{attribute 'no_explicit_call' := 'do not call this FB directly'}{attribute 'enable_dynamic_creation'}
FUNCTION_BLOCK OutputPort_ANY EXTENDS Disposable IMPLEMENTS I_OutputPort
VAR
	_name : T_MAXSTRING;
	_dataType : T_MAXSTRING;
	internalBuffer : POINTER TO BYTE;
	internalBufferSize : UDINT;
	eventEmitter : EventEmitter;
END_VAR

METHOD PUBLIC Accept
VAR_INPUT
	Visitor : I_OutputPortVisitor;
END_VAR
Visitor.VisitOutputPort(this^);
END_METHOD

METHOD PRIVATE CopyInternalBufferToDestination
VAR_INPUT
	DestinationAddress : PVOID;
END_VAR
memcpy(DestinationAddress,internalBuffer,internalBufferSize);
END_METHOD

METHOD PRIVATE CopySourceToInternalBuffer
VAR_INPUT
	SourceAddress : PVOID;
END_VAR
memcpy(internalBuffer,SourceAddress,internalBufferSize);
END_METHOD

PROPERTY PUBLIC DataSize : UDINT
GET
IF internalBuffer = 0 THEN
	RETURN;
END_IF

DataSize := internalBufferSize;
END_GET
END_PROPERTY

PROPERTY PUBLIC DataType : T_MAXSTRING
GET
DataType := _dataType;
END_GET
END_PROPERTY

METHOD PRIVATE DeleteInternalBuffer
IF internalBuffer <> 0 THEN
	__DELETE(internalBuffer);
END_IF
END_METHOD

METHOD PRIVATE EmitOnOutputPortChangeEvent
VAR_INPUT
	PortChanged : I_OutputPort;
END_VAR
VAR
	pOutputPortChangeEvent : POINTER TO OutputPortChangedEvent;
END_VAR
pOutputPortChangeEvent := __NEW(OutputPortChangedEvent(TargetOutputPort := PortChanged));
eventEmitter.Emit('OnOutputPortChanged',pOutputPortChangeEvent^);
pOutputPortChangeEvent^.Dispose();
END_METHOD

METHOD FB_exit : BOOL
VAR_INPUT
	bInCopyCode : BOOL; // if TRUE, the exit method is called for exiting an instance that is copied afterwards (online change).
END_VAR
IF bInCopyCode THEN
	RETURN;
END_IF

DeleteInternalBuffer();
END_METHOD

METHOD FB_init : BOOL
VAR_INPUT
	bInitRetains : BOOL; // if TRUE, the retain variables are initialized (warm start / cold start)
	bInCopyCode : BOOL;  // if TRUE, the instance afterwards gets moved into the copy code (online change)
	Name : T_MAXSTRING;
	DataType : T_MAXSTRING;
	Parent : I_HaveOutputPorts;
END_VAR
_name := Name;
_dataType := DataType;

IF Parent = 0 THEN
	RETURN;
END_IF

Parent.AddOutputPort(THIS^);
END_METHOD

METHOD PUBLIC Get
VAR_INPUT
	Value : ANY;
END_VAR
GetTo(Value.pValue, DINT_TO_UDINT(Value.diSize));
END_METHOD

METHOD PUBLIC GetTo
VAR_INPUT
	Destination : PVOID;
	DestinationSize : UDINT;
END_VAR
IF NOT IsInternalBufferSameSizeAs(DestinationSize) THEN
	RETURN;
END_IF

CopyInternalBufferToDestination(Destination);
END_METHOD

PROPERTY HasData : BOOL
GET
HasData := internalBuffer <> 0 and internalBufferSize <> 0;
END_GET
END_PROPERTY

METHOD PRIVATE IsInternalBufferSameSizeAs : BOOL
VAR_INPUT
	Size : UDINT;
END_VAR
IF internalBuffer = 0 THEN
	RETURN;
END_IF

IF internalBufferSize <> Size THEN
	RETURN;
END_IF

IsInternalBufferSameSizeAs := TRUE;
END_METHOD

METHOD PRIVATE MakeInternalBufferOfSize
VAR_INPUT
	Size : UDINT;
END_VAR
internalBufferSize := Size;
internalBuffer := __NEW(BYTE, internalBufferSize);
END_METHOD

PROPERTY PUBLIC Name : T_MAXSTRING
GET
Name := _name;
END_GET
END_PROPERTY

METHOD PUBLIC OffEvent
VAR_INPUT
	EventName : T_MaxString;
	EventHandler : I_EventHandler;
END_VAR
eventEmitter.OffEvent(EventName, EventHandler);
END_METHOD

METHOD PUBLIC OnceEvent
VAR_INPUT
	EventName : T_MaxString;
	EventHandler : I_EventHandler;
END_VAR
eventEmitter.OnceEvent(EventName, EventHandler);
END_METHOD

METHOD PUBLIC OnEvent
VAR_INPUT
	EventName : T_MaxString;
	EventHandler : I_EventHandler;
END_VAR
eventEmitter.OnEvent(EventName, EventHandler);
END_METHOD

METHOD PUBLIC Set
VAR_INPUT
	Value : ANY;
END_VAR
SetFrom(Value.pValue, DINT_TO_UDINT(Value.diSize));
END_METHOD

METHOD PUBLIC SetFrom
VAR_INPUT
	SourceAddress : PVOID;
	SourceSize : UDINT;
END_VAR
DeleteInternalBuffer();
MakeInternalBufferOfSize(SourceSize);
CopySourceToInternalBuffer(SourceAddress);
EmitOnOutputPortChangeEvent(this^);
END_METHOD

END_FUNCTION_BLOCK

(* stored: Version 1.1.0.1, ProductVersion 3.1.4024.12
   POU OutputPort_ANY: Id {4c7e0bce-9eb0-0f6a-044f-6a3cfc8b783d}, SpecialFunc None
   Folder Constructor: Id {677256cd-e8af-081b-2804-5689f5f4149b}
   Folder Destructor: Id {98956262-b478-014c-3a4b-e5a55f558cc8}
   Folder Private: Id {6f5f4b13-ef19-01e5-075e-0ea3b801d3d7}
   Method Accept: Id {685a8b40-a5b2-0491-3a06-acbf37dad5a1}
   Method CopyInternalBufferToDestination: Id {7ebcbeb6-b02d-0411-1889-2e34c4062c87}
   Method CopySourceToInternalBuffer: Id {dfe21f9e-a5b4-027e-1e44-3be7358a5e65}
   Property DataSize: Id {7a8abb9b-e67f-0be5-36ec-3437e6158ced}
   Get Get: Id {1762b04d-6048-02f1-27c3-298a0a2eb6a2}
   Property DataType: Id {eb163034-b0fd-0fe3-0fa5-fd0220399dfb}
   Get Get: Id {7534416c-ca26-06ef-2b8b-0ad13dd0d8f6}
   Method DeleteInternalBuffer: Id {d61f4872-b9ca-0743-3d16-144280366585}
   Method EmitOnOutputPortChangeEvent: Id {4cedd9f2-3d84-035e-18ce-b7ebc3af2524}
   Method FB_exit: Id {dad2c4bc-10fa-09e1-1929-9db4c4aa6f25}
   Method FB_init: Id {1ba1d2d7-341d-0e8e-05ef-f5346255db4e}
   Method Get: Id {d7f053a1-edb3-045f-2e85-d7d160cdb265}
   Method GetTo: Id {6e5c850e-5dc7-0ca4-0094-d63313848019}
   Property HasData: Id {4031d1bf-7fc9-0b4f-1821-1051bd3aca54}
   Get Get: Id {b11abb15-38ab-0cf1-0107-22a33b095416}
   Method IsInternalBufferSameSizeAs: Id {200fc8fe-6281-0aa7-2e38-670988812e63}
   Method MakeInternalBufferOfSize: Id {d976a026-eec1-07cb-2e0e-d0646f2868ef}
   Property Name: Id {a6251d93-37b5-06d7-00eb-bc1261f23075}
   Get Get: Id {66530c4b-9811-0535-0d83-3db73e2195f3}
   Method OffEvent: Id {5f0c98a6-efae-06ce-0d53-00d24017a360}
   Method OnceEvent: Id {33aa55e6-cc64-0804-1f68-fe127e9ffd59}
   Method OnEvent: Id {83584882-e2df-000f-0211-5ef5ee02b990}
   Method Set: Id {1e1c2da9-f2e1-0401-2df7-d89f92cc9a3e}
   Method SetFrom: Id {76d02626-79e8-0585-25de-a6810fcf20bc} *)
